{attribute 'hide'}
FUNCTION LrealFromBits : LREAL
VAR_INPUT
  b : ULINT;
END_VAR
VAR
  x : POINTER TO LREAL := ADR(b);
END_VAR

LrealFromBits := x^;

END_FUNCTION

(* stored: Version 1.1.0.1
   POU LrealFromBits: Id {26af1350-f1f7-4775-a258-be47fc01563f}, SpecialFunc None *)
